{attribute 'GeneratedUsingTerminal: Flexi Gateway GETC1-0001-0000'}
{attribute addProperty BoxType "Flexi Gateway GETC1-0001-0000"}
{attribute addProperty Id "New_Messages_AvailableAT %I*BOOL1"}
{attribute addProperty CRC "1434060703"}
{attribute addProperty Size "1"}
TYPE NewMessageFlag_557A079F EXTENDS TcoIo.InputBase_8311D824 :
STRUCT
	{attribute addProperty Name "New_Messages_Available"}
	New_Messages_Available AT %I* : BOOL;
END_STRUCT
END_TYPE

(* stored: Version 1.2.0.0, ProductVersion 3.1.4024.11
   DUT NewMessageFlag_557A079F: Id {aff608df-9942-03a5-12b5-015159f7c59a} *)
